Fanuc KAREL source: ko00048.KL

-- PROVISIONAL review KL for V1013-1; original PC SHA256 a00af6273f3e36a27189f7475f66b3a5c63ebd827e8671548153de5a1b4cb4bb
-- Incomplete behavior may be omitted. Consult companion uncertainty JSON. Do not deploy.
PROGRAM KO00048
%NOLOCKGROUP
BEGIN
  -- UNRESOLVED_PC offsets 5-12; opcodes 9D,23
  -- UNRESOLVED_PC offsets 17-69; opcodes 27,27,49,7E,AD,27,49,7E,AD,22,31,7E,4A
  -- UNRESOLVED_PC offsets 74-78; opcodes 7F
END KO00048
